{attribute 'linkalways'} 
{attribute 'no_explicit_call' := 'This FB is a CLASS and must be accessed using methods or properties'}
{attribute 'enable_dynamic_creation'}
FUNCTION_BLOCK FINAL SUB_UDINT EXTENDS Node
VAR
	in1 : _UDINT(0);
	in2 : _UDINT(0);
	out : _UDINT(0);
END_VAR

METHOD PUBLIC Clone : I_Node
VAR
	pNode : POINTER TO SUB_UDINT;
END_VAR
pNode := __NEW(SUB_UDINT);
Clone := pNode^;
END_METHOD

METHOD FB_init : BOOL
VAR_INPUT
	bInitRetains : BOOL; // if TRUE, the retain variables are initialized (warm start / cold start)
	bInCopyCode : BOOL;  // if TRUE, the instance afterwards gets moved into the copy code (online change)
END_VAR
AddInput('in1',THIS^.in1);
AddInput('in2',THIS^.in2);
AddOutput('out', THIS^.out);
END_METHOD

METHOD PROTECTED OnExecute
VAR
END_VAR
out.Value := in1.Value - in2.Value;
END_METHOD

END_FUNCTION_BLOCK

(* stored: Version 1.1.0.1, ProductVersion 3.1.4024.15
   POU SUB_UDINT: Id {0c2c5ae6-9c89-4db7-8a83-380d71ef4b6c}, SpecialFunc None
   Folder Constructor: Id {55699c79-4b1d-46c3-af05-8077d333ebec}
   Method Clone: Id {a8476edc-9702-4aed-8a32-ee7f58360bff}
   Method FB_init: Id {fe392a00-5453-4ea3-aca3-0b0677a9c9f1}
   Method OnExecute: Id {1406e7b5-52e5-4c3f-ae9c-8cebfcb37a2a} *)
